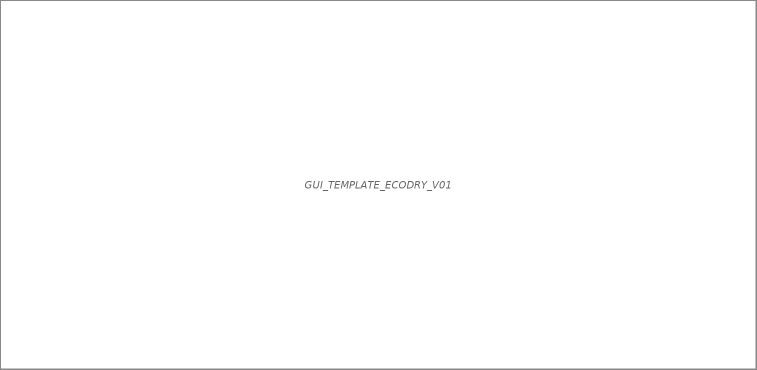
VISUALIZATION GUI_ECODRY_V01_EVAC_LAB  // 757x370
    Frame (0,0 757x370)
        shows GUI_TEMPLATE_ECODRY_V01(m_Instance := MAIN.evac_lab.rp, m_bEnable := MAIN.evac_lab.ctrl.bEnable_RP)
END_VISUALIZATION

(* stored: Version 1.1.0.1, ProductVersion 3.1.4024.9
   Visu GUI_ECODRY_V01_EVAC_LAB: Id {a212054e-3367-4d17-973b-8d4390b7b313} *)
